FUNCTION_BLOCK NotificationCollection IMPLEMENTS Collection
VAR
	numberOfItems 			: INT := 0;
	pNotificationList 		: ARRAY[0..Param.MAX_ITERABLE_ITEMS] OF POINTER TO Notification;
	pNotificationIterator 	: POINTER TO NotificationIterator;
END_VAR

METHOD addItem
VAR_INPUT
	str : STRING;
END_VAR
IF (THIS^.numberOfItems >= Param.MAX_ITERABLE_ITEMS) THEN
	ADSLOGSTR( msgCtrlMask := ADSLOG_MSGTYPE_ERROR, msgFmtStr := 'PLC Msg. : %s', strArg := 'System Full');
ELSE
	THIS^.pNotificationList[THIS^.numberOfItems] := __NEW(Notification(sNotification := str));
	THIS^.numberOfItems := THIS^.numberOfItems + 1;
END_IF
END_METHOD

METHOD createIterator : Iterator
THIS^.pNotificationIterator := __NEW(NotificationIterator(pNotificationList := THIS^.pNotificationList));
createIterator := THIS^.pNotificationIterator^;
END_METHOD

METHOD FB_exit : BOOL
VAR_INPUT
	bInCopyCode : BOOL; // if TRUE, the exit method is called for exiting an instance that is copied afterwards (online change).
END_VAR

VAR
	i: INT;
END_VAR
FOR i:=0 TO Param.MAX_ITERABLE_ITEMS DO
	IF THIS^.pNotificationList[i] <> 0 THEN
		__DELETE(THIS^.pNotificationList[i]);
	END_IF
END_FOR

IF THIS^.pNotificationIterator <> 0 THEN
	__DELETE(THIS^.pNotificationIterator);
END_IF
END_METHOD

METHOD FB_init : BOOL
VAR_INPUT
	bInitRetains : BOOL; // if TRUE, the retain variables are initialized (warm start / cold start)
	bInCopyCode : BOOL;  // if TRUE, the instance afterwards gets moved into the copy code (online change)
END_VAR
END_METHOD

END_FUNCTION_BLOCK

(* stored: Version 1.1.0.1, ProductVersion 3.1.4024.12
   POU NotificationCollection: Id {6cb89627-31bd-4642-8a55-4b368ad29f85}, SpecialFunc None
   Method addItem: Id {849580a8-5029-457b-81ec-32062fadb444}
   Method createIterator: Id {1217f06b-3955-47d7-8a5c-0fa572fc7931}
   Method FB_exit: Id {9ed9e0be-83a5-4a20-9cd8-116735871b38}
   Method FB_init: Id {bc95b514-aece-4f53-ae16-4ba63c2bc5fb} *)
